// TIA Portal V19 export
DATA_BLOCK "SeqData"   // DB11
TITLE = SeqData
{ S7_Optimized_Access := 'TRUE'; DB_Accessible_From_OPC_UA := 'FALSE' }
AUTHOR : Siemens
// Global DB for BeltLift
// stored: DBAccessibleFromOPCUA false, MemoryReserve 100
   VAR
      plantOn : Bool := true;   // Plant switched on
      compressedAir : Bool;   // Druckluft nicht in Ordnung. Im Fehlerfall ist die Ursache: Der zur Maschine gehörende Not-Halt hat die Maschine gestoppt. Bei ausgeschalteter Maschine oder gedrücktem Not-Halt können keine Funktionen ausgeführt werden. / Compressed air not OK. In case of an Error Cause: The emergency stop belonging to the machine has stopped the machine. No functions can be performed when the machine is shut off or the emergency stop is pressed.
      powerVoltage : Bool;   // Spannungsversorgung nicht in Ordnung. Im Fehlerfall ist die Druckluft nicht in Ordnung. Im Fehlerfall ist die Ursache: Der zur Maschine gehörende Not-Halt hat die Maschine gestoppt. Bei ausgeschalteter Maschine oder gedrücktem Not-Halt können keine Funktionen ausgeführt werden. / Voltage power supply not OK.
      doorClosed : Bool;   // Safety door closed
      autoStart : Bool;   // Automatic start
      autoStop : Bool;   // Automatic stop
      autoStarted : Bool := false;   // Automatic started
      autoStopped : Bool;   // Automatic stopped
      ackSeq : Bool;   // Acknowledge GRAPH FB
      errFltSeq : Bool;   // Error Graph FB
      seqStart : Bool;   // GRAPH sequence started
      newCase : Bool;   // Sensor new case
      posCaseBelt : Int;   // Case position on belt
      posLift1 : Int;   // Lift 1 position
      posLift2 : Int;   // Lift 2 position
      visCaseLift1 : Bool;   // Case lift1 visible
      visCaseLift2 : Bool;   // Case lift2 visible
      setStop1 : Bool;   // Set stopper1
      setStop2 : Bool;   // Set stopper2
      sensorStop1 : Bool;   // Sensor at stopper1
      sensorStop2 : Bool;   // Sensor at stopper2
      sensorStop3 : Bool;   // Sensor at stopper3
      errSensorStop1 : Bool;   // Error on Sensor at stopper1
      errSensorStop2 : Bool;   // Error on Sensor at stopper2
      errSensorStop3 : Bool;   // Error on Sensor at stopper2
      errSensorNewCase : Bool;   // Error on Sensor at new case
      toLift1 : Bool;   // Case to lift1 or lift2
      autoLift1 : "typeStartLift";   // Start automatic lift1
      autoLift2 : "typeStartLift";   // Start automatic lift2
      manLift1 : "typeStartLift";   // Start manual lift1
      manLift2 : "typeStartLift";   // Start manual lift2
      outLift1Up : Bool;   // Output lift1 up
      outLift1Down : Bool;   // Output lift1 down
      outLift2Up : Bool;   // Output lift2 up
      outLift2Down : Bool;   // Output lift2 down
      sensorLift1Up : Bool;   // Sensor lift1 up
      sensorLift1Down : Bool;   // Sensor lift1 down
      sensorLift2Up : Bool;   // Sensor lift2 up
      sensorLift2Down : Bool;   // Sensor lift2 down
      simOperandSupVis : Bool;   // Simulation supervision operand
      simInterlockSupVis : Bool;   // Simulation supervision interlock
      simLiftFreeSupVis : Bool;   // Simulation supervision lift free
      simActReactSupVis : Bool;   // Simulation supervision action and reaction
      simPositionSupVis : Bool;   // Simulation supervision position
      simUdtOperandSupVis : Bool;   // Simulation supervision operand in UDT
      simActive : Bool;   // Simulation active
      releaseSimPlantOn : Bool;   // Release simulation plant on
      releaseSimAutoStarted : Bool;   // Release simulation auto started
      releaseSimAutoStopped : Bool;   // Release simulation auto stopped
      beltLEDs : Word;   // Moving lights belt
      lift1LEDs : Word;   // Moving lights lift1
      lift2LEDs : Word;   // Moving lights lift2
      stateCase : Array[0..3] of Bool;   // State case position
      liftFree : Bool := true;   // Lift is free for new case / Lift ist bereit für einen neuen Kasten
      simInterlockSupVisLiftFree : Bool;   // Simulation supervision interlock / Simulation supervision interlock lift free
      resetCrit : Bool;
      identTimeStamp : LDT;
      retVal : Int;
      frequency : Real := 10.0;
      freqError : Bool;
      freqStatus : Word;
      textListID { ExternalAccessible := 'False'; ExternalVisible := 'False'; ExternalWritable := 'False'} : Word;
   END_VAR
BEGIN
END_DATA_BLOCK
